// Mitsubishi GX Works2 project: Group19_plc_run   PLC: FX3G

// global labels: Global1
VAR_GLOBAL
  startday AT X007 : BOOL;
END_VAR
VAR_GLOBAL CONSTANT
  ShmarimInput : INT := 300;
END_VAR
VAR_GLOBAL
  ShmarimQuantity AT D1117 : INT;
  MinShmarim AT D1119 : INT;
END_VAR
VAR_GLOBAL CONSTANT
  LetetInput : INT := 20;
END_VAR
VAR_GLOBAL
  LetetQuantity AT D1121 : INT;
END_VAR
VAR_GLOBAL CONSTANT
  KashutInput : INT := 130;
END_VAR
VAR_GLOBAL
  KashutQuantity AT D1125 : INT;
  Lamp7 AT Y007 : BOOL;
  Check1 AT X001 : BOOL;
  CheckAnalogInput1 AT X001 : BOOL;
  ifLagerBeer AT M16 : BOOL;
END_VAR
VAR_GLOBAL CONSTANT
  Five : INT := 5;
END_VAR
VAR_GLOBAL
  FlinzerBeer AT M18 : BOOL;
END_VAR
VAR_GLOBAL CONSTANT
  MinmumShmarimLager : INT := 150;
END_VAR
VAR_GLOBAL
  EndDay AT M10 : BOOL;
  ifShmarimQuantityEnoughToLager AT M20 : BOOL;
END_VAR
VAR_GLOBAL CONSTANT
  MinmumLetetLager : INT := 12;
END_VAR
VAR_GLOBAL
  ifLetetQuantityEnoughToLager AT M22 : BOOL;
  KashotQuantity AT D1125 : INT;
END_VAR
VAR_GLOBAL CONSTANT
  MinmumKashotLager : INT := 60;
END_VAR
VAR_GLOBAL
  ifKashotQuantityEnoughToLager AT M24 : BOOL;
  Label20 AT M20 : BOOL;
  Label22 AT M22 : BOOL;
  Label1 AT M10 : BOOL;
  Label12 AT M12 : BOOL;
  Label10 AT M120 : BOOL;
  Label14 AT M14 : BOOL;
  TimerCook AT E4 : REAL;
END_VAR
VAR_GLOBAL CONSTANT
  AnalogDivide : INT := 400;
  MinmumShmarimFlinzer : INT := 120;
  MinmumLetetFlinzer : INT := 6;
  MinmumKashotFlinzer : INT := 54;
END_VAR
VAR_GLOBAL
  ifShmarimQuantityEnoughToFlinzer AT M26 : BOOL;
  ifLetetQuantityEnoughToFlinzer AT M28 : BOOL;
  ifKashotQuantityEnoughToFlinzer AT M30 : BOOL;
END_VAR
VAR_GLOBAL CONSTANT
  TimerCook4 : INT := 40;
END_VAR
VAR_GLOBAL
  CookBeer AT Y001 : BOOL;
  TempLamp4 AT M32 : BOOL;
  AfterCook4Sec AT Y001 : BOOL;
  EndOfCooking AT M62 : BOOL;
  After5Sec AT TS1 : BOOL;
  startTransferBeer AT X005 : BOOL;
  FlickerLager1 AT M36 : BOOL;
  TS2 AT TS2 : BOOL;
  labelTS2 AT TS2 : BOOL;
  labelTS3 AT TS3 : BOOL;
  Lamp3 AT Y003 : BOOL;
  TC4 : BOOL;
  labelTC2 AT TC2 : BOOL;
  labelTC3 AT TC3 : BOOL;
  labelTC4 AT TC4 : BOOL;
  labelTS4 AT TS4 : BOOL;
  Lamp4 AT Y004 : BOOL;
  labelTC5 AT TC5 : BOOL;
  labelTS5 AT TS5 : BOOL;
  labelTC6 AT TC6 : BOOL;
  labelTS6 AT TS6 : BOOL;
  FlickerFlinzer1 AT M38 : BOOL;
  labelTC7 AT TC7 : BOOL;
  labelTS7 AT TS7 : BOOL;
  AfterFlicker AT X002 : BOOL;
  PutOneBeer AT X000 : BOOL;
  CounterFirst AT CC1 : BOOL;
END_VAR
VAR_GLOBAL CONSTANT
  CounterOne : INT := 1;
END_VAR
VAR_GLOBAL
  StartPackging AT M40 : BOOL;
  CounterSecond AT CC2 : BOOL;
END_VAR
VAR_GLOBAL CONSTANT
  CounterSix : INT := 6;
END_VAR
VAR_GLOBAL
  OpenLightAfterOneBeer AT CS1 : BOOL;
  OneBeerIn AT Y002 : BOOL;
  CloseLightAfter6Beers AT CS2 : BOOL;
  CounterSixPacks AT D1127 : INT;
END_VAR
VAR_GLOBAL CONSTANT
  AddOneSix : INT := 1;
  TimerTsisaLager : INT := 30;
  TimerTsisaFlicker : INT := 40;
END_VAR
VAR_GLOBAL
  TC_1 AT TC1 : BOOL;
  TC_2 AT TC2 : BOOL;
  TC_3 AT TC3 : BOOL;
  TC_4 AT TC4 : BOOL;
END_VAR
VAR_GLOBAL CONSTANT
  TimerTsisaFlinser : INT := 40;
END_VAR
VAR_GLOBAL
  FinishDay AT X011 : BOOL;
  AnalogInput AT D8280 : INT;
  startflickeringLager AT M42 : BOOL;
  startflicker AT M44 : BOOL;
  labelTS1 AT TS1 : BOOL;
  HelpLamp AT M60 : BOOL;
  TC_9_outOfFlikering AT TC9 : BOOL;
  EndOfFlickering100 AT M64 : BOOL;
  TC9Out AT TC9 : BOOL;
  HelpLamp2 AT M64 : BOOL;
  HelpLamp3 AT M66 : BOOL;
END_VAR
VAR_GLOBAL CONSTANT
  TimerTsisaLager1 : INT := 30;
END_VAR
VAR_GLOBAL
  labelTS9 AT TS9 : BOOL;
END_VAR
VAR_GLOBAL CONSTANT
  TimerTsisaLager_flickering : INT := 5;
END_VAR
VAR_GLOBAL
  TC10 AT TC10 : BOOL;
  labelTC10 AT TC10 : BOOL;
  labelTS10 AT TS10 : BOOL;
  labelTC_5 AT TC5 : BOOL;
  startflickeringFlinzer AT M80 : BOOL;
  HelpLampPackging AT M90 : BOOL;
  Track AT CN2 : INT;
  Try AT CN2 : INT;
  Label_Iteration AT M84 : BOOL;
  AnalogOutput AT D8282 : INT;
  new_sixPack AT M86 : BOOL;
END_VAR
VAR_GLOBAL CONSTANT
  Min_ShmarimLager : REAL := 150;
  Min_LetetLager : REAL := 12;
  Min_KashutLager : REAL := 60;
  Min_ShmarimFilzner : REAL := 120;
  Min_LetetFilzner : REAL := 6;
  Min_KashutFilzner : REAL := 54;
END_VAR

// task Task_01 (event TRUE, interval 0, priority 31): POU_01

PROGRAM POU_01
(* structured ladder/FBD written out as ST: instructions are called as NAME(EN, inputs, outputs); _pN, _eN, _tN stand for wires *)
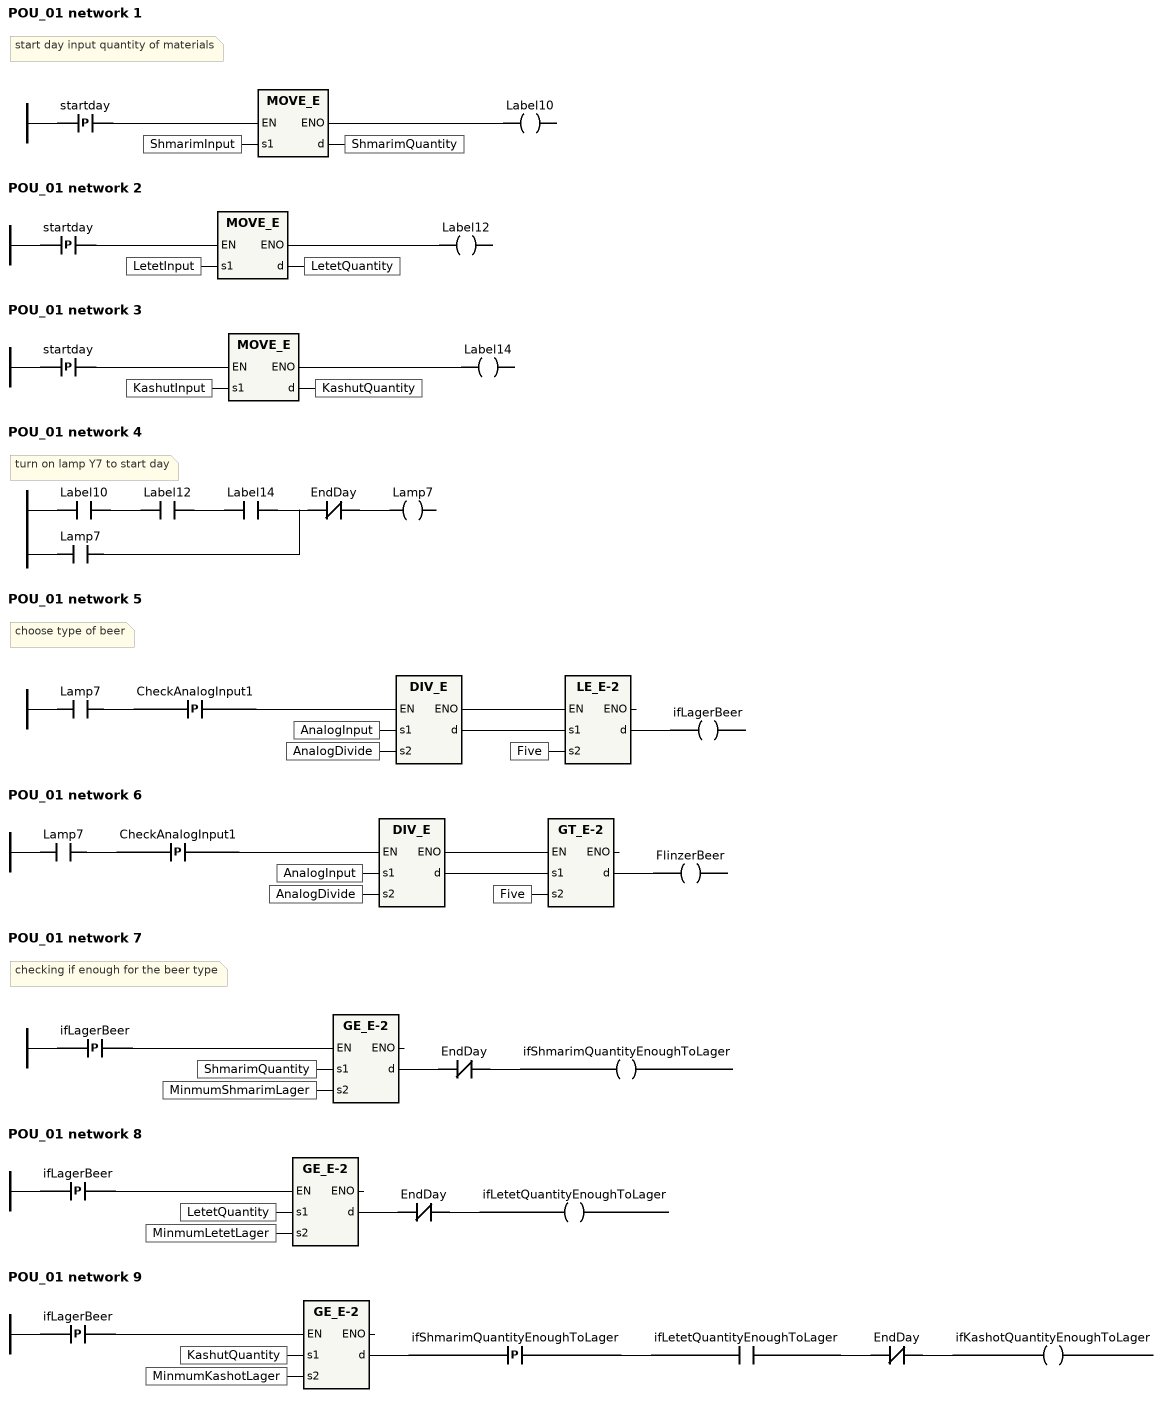
(* network 1 *)
(* start day input quantity of materials *)
_e1 := MOVE_E(LDP(TRUE, startday), ShmarimInput, ShmarimQuantity);
Label10 := _e1;
(* network 2 *)
_e1 := MOVE_E(LDP(TRUE, startday), LetetInput, LetetQuantity);
Label12 := _e1;
(* network 3 *)
_e1 := MOVE_E(LDP(TRUE, startday), KashutInput, KashutQuantity);
Label14 := _e1;
(* network 4 *)
(* turn on lamp Y7 to start day *)
Lamp7 := ((Label10 AND Label12 AND Label14) OR Lamp7) AND NOT EndDay;
(* network 5 *)
(* choose type of beer *)
_e2 := DIV_E(Lamp7 AND LDP(TRUE, CheckAnalogInput1), AnalogInput, AnalogDivide, _t1);
LE_E(_e2, _t1, Five, _t3);
ifLagerBeer := _t3;
(* network 6 *)
_e2 := DIV_E(Lamp7 AND LDP(TRUE, CheckAnalogInput1), AnalogInput, AnalogDivide, _t1);
GT_E(_e2, _t1, Five, _t3);
FlinzerBeer := _t3;
(* network 7 *)
(* checking if enough for the beer type *)
GE_E(LDP(TRUE, ifLagerBeer), ShmarimQuantity, MinmumShmarimLager, _t1);
ifShmarimQuantityEnoughToLager := _t1 AND NOT EndDay;
(* network 8 *)
GE_E(LDP(TRUE, ifLagerBeer), LetetQuantity, MinmumLetetLager, _t1);
ifLetetQuantityEnoughToLager := _t1 AND NOT EndDay;
(* network 9 *)
GE_E(LDP(TRUE, ifLagerBeer), KashutQuantity, MinmumKashotLager, _t1);
ifKashotQuantityEnoughToLager := _t1 AND LDP(TRUE, ifShmarimQuantityEnoughToLager) AND ifLetetQuantityEnoughToLager AND NOT EndDay;
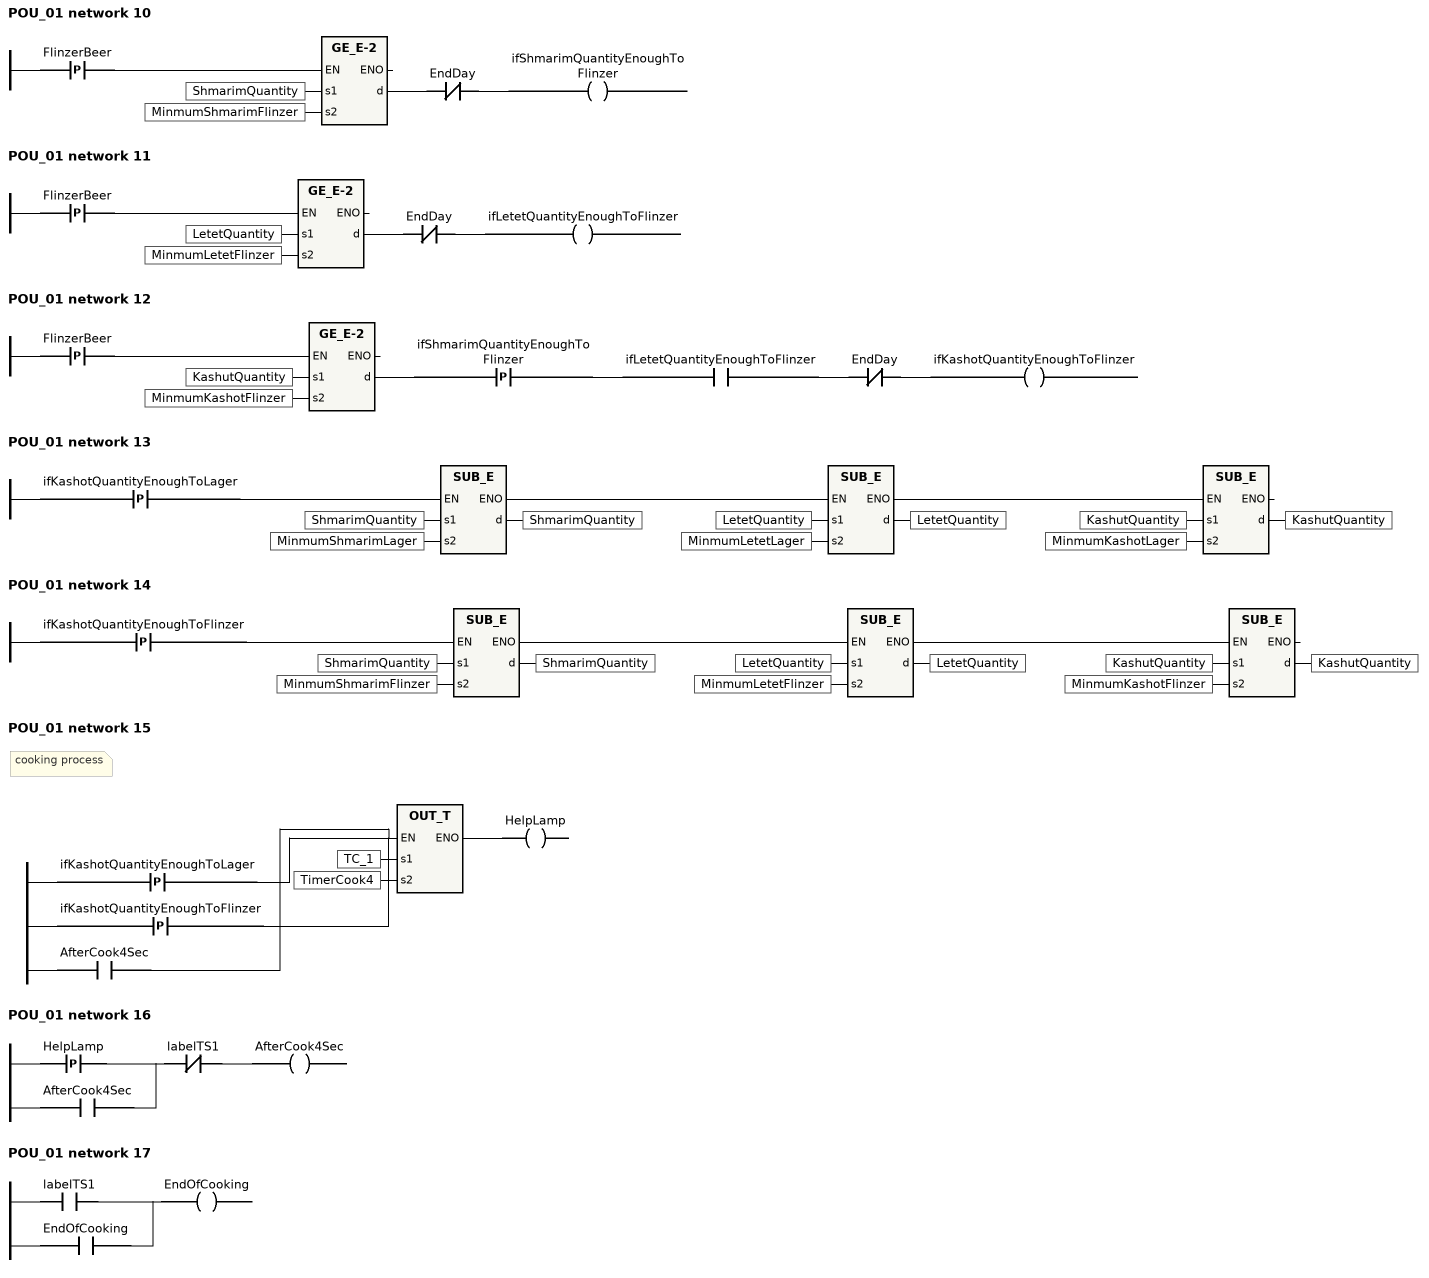
(* network 10 *)
GE_E(LDP(TRUE, FlinzerBeer), ShmarimQuantity, MinmumShmarimFlinzer, _t1);
ifShmarimQuantityEnoughToFlinzer := _t1 AND NOT EndDay;
(* network 11 *)
GE_E(LDP(TRUE, FlinzerBeer), LetetQuantity, MinmumLetetFlinzer, _t1);
ifLetetQuantityEnoughToFlinzer := _t1 AND NOT EndDay;
(* network 12 *)
GE_E(LDP(TRUE, FlinzerBeer), KashutQuantity, MinmumKashotFlinzer, _t1);
ifKashotQuantityEnoughToFlinzer := _t1 AND LDP(TRUE, ifShmarimQuantityEnoughToFlinzer) AND ifLetetQuantityEnoughToFlinzer AND NOT EndDay;
(* network 13 *)
_e1 := SUB_E(LDP(TRUE, ifKashotQuantityEnoughToLager), ShmarimQuantity, MinmumShmarimLager, ShmarimQuantity);
_e2 := SUB_E(_e1, LetetQuantity, MinmumLetetLager, LetetQuantity);
SUB_E(_e2, KashutQuantity, MinmumKashotLager, KashutQuantity);
(* network 14 *)
_e1 := SUB_E(LDP(TRUE, ifKashotQuantityEnoughToFlinzer), ShmarimQuantity, MinmumShmarimFlinzer, ShmarimQuantity);
_e2 := SUB_E(_e1, LetetQuantity, MinmumLetetFlinzer, LetetQuantity);
SUB_E(_e2, KashutQuantity, MinmumKashotFlinzer, KashutQuantity);
(* network 15 *)
(* cooking process *)
_e1 := OUT_T(LDP(TRUE, ifKashotQuantityEnoughToLager) OR LDP(TRUE, ifKashotQuantityEnoughToFlinzer) OR AfterCook4Sec, TC_1, TimerCook4);
HelpLamp := _e1;
(* network 16 *)
AfterCook4Sec := (LDP(TRUE, HelpLamp) OR AfterCook4Sec) AND NOT labelTS1;
(* network 17 *)
EndOfCooking := labelTS1 OR EndOfCooking;
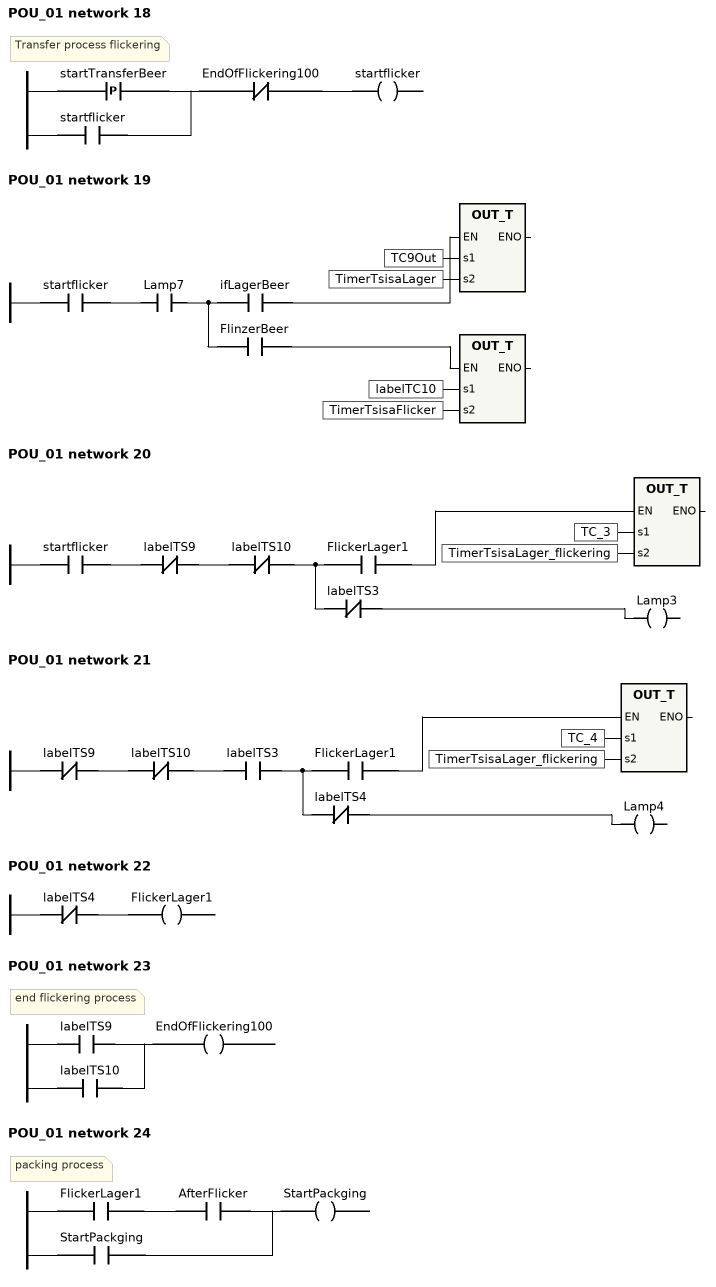
(* network 18 *)
(* Transfer process flickering *)
startflicker := (LDP(TRUE, startTransferBeer) OR startflicker) AND NOT EndOfFlickering100;
(* network 19 *)
_p1 := startflicker AND Lamp7;
OUT_T(_p1 AND ifLagerBeer, TC9Out, TimerTsisaLager);
OUT_T(_p1 AND FlinzerBeer, labelTC10, TimerTsisaFlicker);
(* network 20 *)
_p1 := startflicker AND NOT labelTS9 AND NOT labelTS10;
OUT_T(_p1 AND FlickerLager1, TC_3, TimerTsisaLager_flickering);
Lamp3 := _p1 AND NOT labelTS3;
(* network 21 *)
_p1 := NOT labelTS9 AND NOT labelTS10 AND labelTS3;
OUT_T(_p1 AND FlickerLager1, TC_4, TimerTsisaLager_flickering);
Lamp4 := _p1 AND NOT labelTS4;
(* network 22 *)
FlickerLager1 := NOT labelTS4;
(* network 23 *)
(* end flickering process *)
EndOfFlickering100 := labelTS9 OR labelTS10;
(* network 24 *)
(* packing process *)
StartPackging := (FlickerLager1 AND AfterFlicker) OR StartPackging;
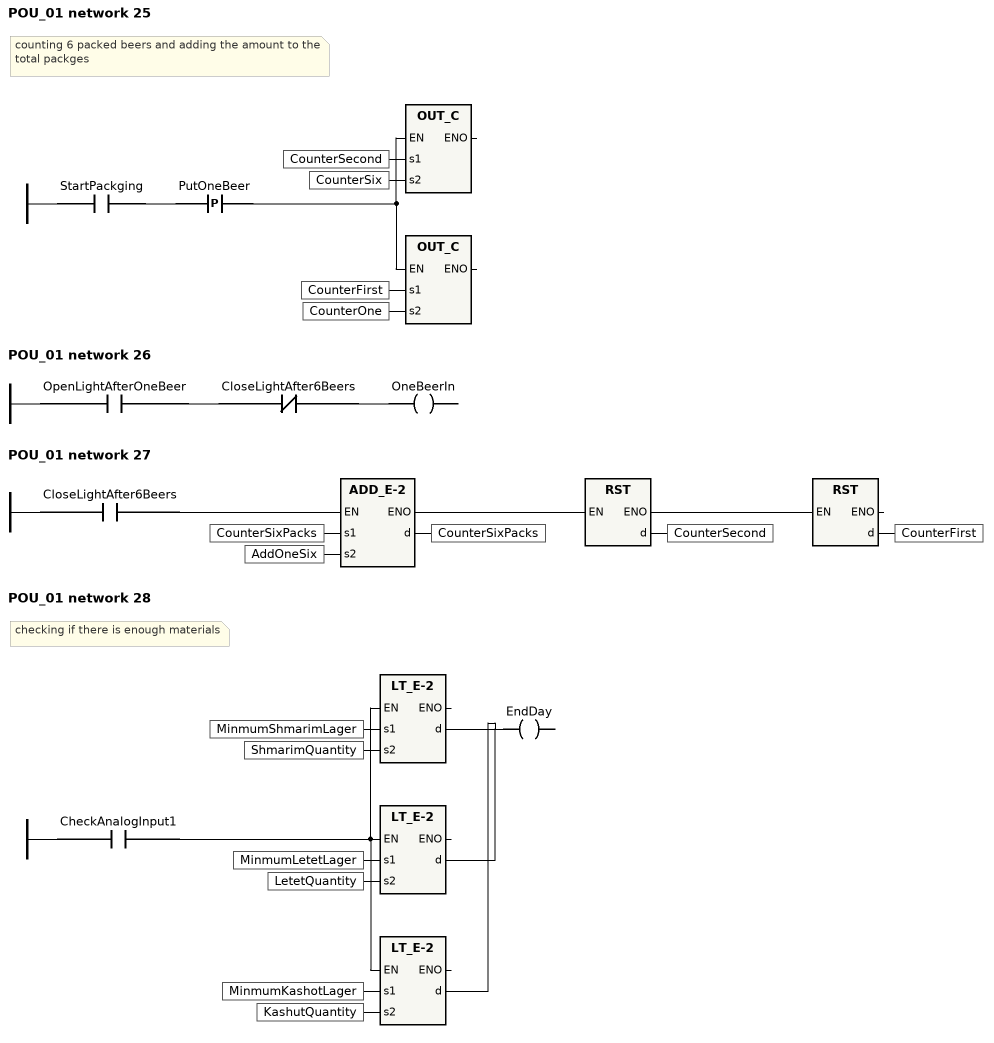
(* network 25 *)
(* counting 6 packed beers and adding the amount to the total packges *)
_p1 := StartPackging AND LDP(TRUE, PutOneBeer);
OUT_C(_p1, CounterSecond, CounterSix);
OUT_C(_p1, CounterFirst, CounterOne);
(* network 26 *)
OneBeerIn := OpenLightAfterOneBeer AND NOT CloseLightAfter6Beers;
(* network 27 *)
_e1 := ADD_E(CloseLightAfter6Beers, CounterSixPacks, AddOneSix, CounterSixPacks);
_e2 := RST(_e1, CounterSecond);
RST(_e2, CounterFirst);
(* network 28 *)
(* checking if there is enough materials *)
LT_E(CheckAnalogInput1, MinmumShmarimLager, ShmarimQuantity, _t1);
LT_E(CheckAnalogInput1, MinmumLetetLager, LetetQuantity, _t2);
LT_E(CheckAnalogInput1, MinmumKashotLager, KashutQuantity, _t3);
EndDay := _t1 OR _t2 OR _t3;
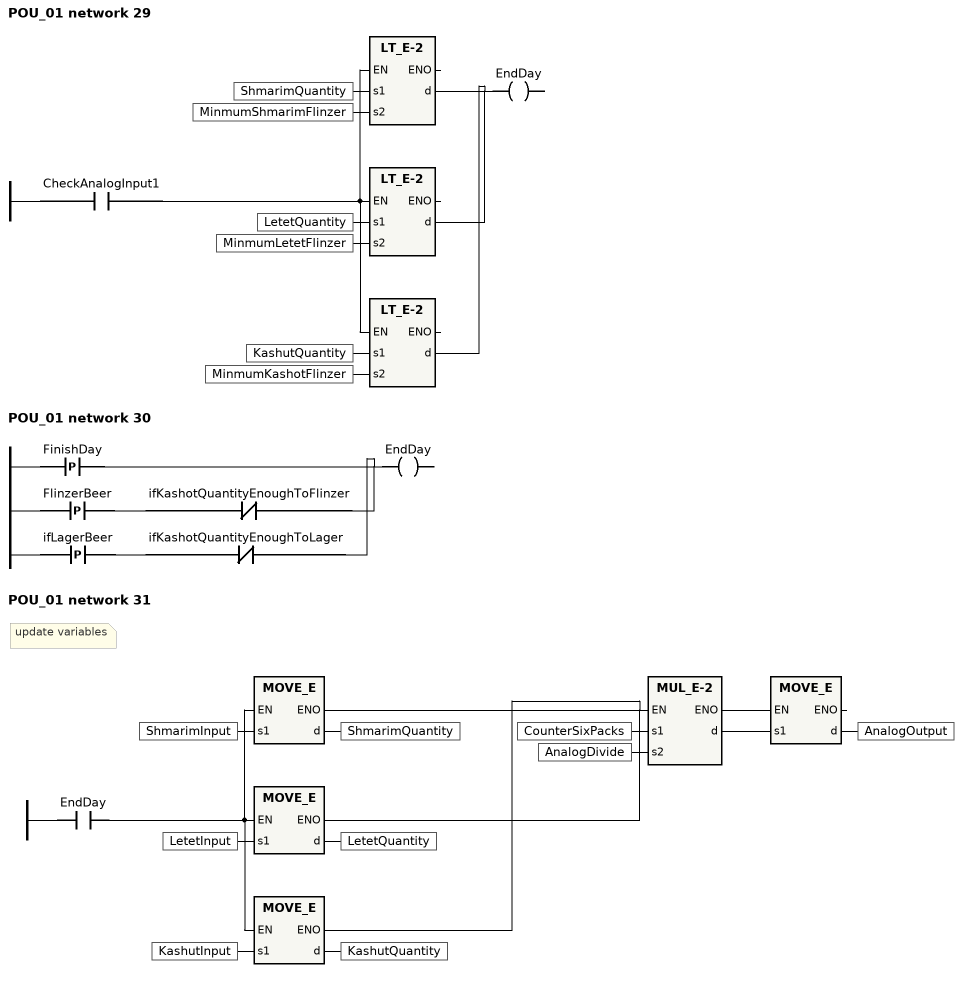
(* network 29 *)
LT_E(CheckAnalogInput1, ShmarimQuantity, MinmumShmarimFlinzer, _t1);
LT_E(CheckAnalogInput1, LetetQuantity, MinmumLetetFlinzer, _t2);
LT_E(CheckAnalogInput1, KashutQuantity, MinmumKashotFlinzer, _t3);
EndDay := _t1 OR _t2 OR _t3;
(* network 30 *)
EndDay := LDP(TRUE, FinishDay) OR (LDP(TRUE, FlinzerBeer) AND NOT ifKashotQuantityEnoughToFlinzer) OR (LDP(TRUE, ifLagerBeer) AND NOT ifKashotQuantityEnoughToLager);
(* network 31 *)
(* update variables *)
_e1 := MOVE_E(EndDay, ShmarimInput, ShmarimQuantity);
_e2 := MOVE_E(EndDay, LetetInput, LetetQuantity);
_e3 := MOVE_E(EndDay, KashutInput, KashutQuantity);
_e5 := MUL_E(_e1 OR _e2 OR _e3, CounterSixPacks, AnalogDivide, _t4);
MOVE_E(_e5, _t4, AnalogOutput);
END_PROGRAM
